// TIA Portal V17 export
// export: Created 2025-03-05T08:02:09.6549569Z, ExportSetting WithDefaults, DisplayName Totally Integrated Automation Portal, DisplayVersion V17 Update 8, DisplayName TIA Portal Openness, DisplayVersion V17 Update 8, DisplayName TIA Portal Version Control Interface, DisplayVersion V17, DisplayName SINAMICS Startdrive Advanced, DisplayVersion V17 SP2, DisplayName SINAMICS Startdrive G110M, G120, G120C, G120D, G120P, G115D, DisplayVersion V17 SP2, DisplayName SINAMICS Startdrive G130, G150, S120, S150, SINAMICS MV, S210, DisplayVersion V17 SP2, DisplayName STEP 7 Professional, DisplayVersion V17 Update 8, DisplayName SINUMERIK ONE STEP 7 Toolbox, DisplayVersion V17 Update 12, DisplayName SINUMERIK 840D sl STEP 7 Toolbox, DisplayVersion V17 Update 12, DisplayName STEP 7 Safety, DisplayVersion V17 Update 6, DisplayName WinCC Advanced, DisplayVersion V17 Update 8
TYPE "TABLE_MAGAZINE"
// stored: IsFailsafeCompliant false
   STRUCT
      NAME_POS : Array[1..60, 1..32] of Char;   // NAME POSITION
      NUM_POS : Array[1..60] of Int;   // NUM POSITION
      PRESENT_POS : Array[1..60] of Bool;   // PRESENT POSITION
      SERIAL_NUMBER : Array[1..60] of DInt;   // SERIAL NUMBER
      TOOL_IN_FAULT : Array[1..60] of Bool;   // TOOL IN FAULT
      WARNING_EDGE1 : Array[1..60] of DInt;   // WARNING EDGE 1
      QUANTITY_EDGE1 : Array[1..60] of DInt;   // QUANTITY EDGE 1
      TOTAL_LIFE_EDGE1 : Array[1..60] of DInt;   // TOTAL LIFE EDGE 1
      WARNING_EDGE2 : Array[1..60] of DInt;   // WARNING EDGE 2
      QUANTITY_EDGE2 : Array[1..60] of DInt;   // QUANTITY EDGE 2
      TOTAL_LIFE_EDGE2 : Array[1..60] of DInt;   // TOTAL LIFE EDGE 2
      WARNING_EDGE3 : Array[1..60] of DInt;   // WARNING EDGE 3
      QUANTITY_EDGE3 : Array[1..60] of DInt;   // QUANTITY EDGE 3
      TOTAL_LIFE_EDGE3 : Array[1..60] of DInt;   // TOTAL LIFE EDGE 3
      WARNING_EDGE4 : Array[1..60] of DInt;   // WARNING EDGE 4
      QUANTITY_EDGE4 : Array[1..60] of DInt;   // QUANTITY EDGE 4
      TOTAL_LIFE_EDGE4 : Array[1..60] of DInt;   // TOTAL LIFE EDGE 4
      WARNING_EDGE5 : Array[1..60] of DInt;   // WARNING EDGE 5
      QUANTITY_EDGE5 : Array[1..60] of DInt;   // QUANTITY EDGE 5
      TOTAL_LIFE_EDGE5 : Array[1..60] of DInt;   // TOTAL LIFE EDGE 5
   END_STRUCT;
END_TYPE
